(* IEC 61131-3 sources: STruCpp/tests/st-validation/function_blocks, 30 files *)

(* ---- basic_fb.st ---- *)
FUNCTION_BLOCK Counter
  VAR_INPUT increment : INT; END_VAR
  VAR_OUTPUT count : INT; END_VAR
  count := count + increment;
END_FUNCTION_BLOCK

FUNCTION_BLOCK Toggle
  VAR_OUTPUT state : BOOL; END_VAR
  state := NOT state;
END_FUNCTION_BLOCK

(* ---- fb_abstract.st ---- *)
FUNCTION_BLOCK ABSTRACT Shape
  VAR_OUTPUT area : REAL; END_VAR

  METHOD PUBLIC ABSTRACT GetArea : REAL
  END_METHOD
END_FUNCTION_BLOCK

FUNCTION_BLOCK Circle EXTENDS Shape
  VAR_INPUT radius : REAL; END_VAR

  METHOD PUBLIC GetArea : REAL
    GetArea := 3.14159 * radius * radius;
  END_METHOD

  area := THIS.GetArea();
END_FUNCTION_BLOCK

(* ---- fb_accumulator.st ---- *)
FUNCTION_BLOCK AccumulatorFB
  VAR_INPUT inc : INT; END_VAR
  VAR total : INT; END_VAR
  VAR_OUTPUT result : INT; END_VAR
  total := total + inc;
  result := total;
END_FUNCTION_BLOCK

(* ---- fb_composition.st ---- *)
FUNCTION_BLOCK Sensor
  VAR_OUTPUT value : INT; END_VAR
  value := 42;
END_FUNCTION_BLOCK

FUNCTION_BLOCK Controller
  VAR
    sensor : Sensor;
    reading : INT;
    processed : BOOL;
  END_VAR
  sensor();
  reading := sensor.value;
  processed := TRUE;
END_FUNCTION_BLOCK

(* ---- fb_constructor_defaults.st ---- *)
FUNCTION_BLOCK ConfigFB
  VAR_INPUT
    maxCount : INT;
  END_VAR
  VAR_OUTPUT
    ready : BOOL;
  END_VAR
  VAR
    counter : INT;
  END_VAR
  IF counter < maxCount THEN
    counter := counter + 1;
  END_IF;
  ready := counter >= maxCount;
END_FUNCTION_BLOCK

(* ---- fb_deep_method.st ---- *)
FUNCTION_BLOCK Inner
  VAR_INPUT seed : INT; END_VAR
  VAR_OUTPUT val : INT; END_VAR
  METHOD PUBLIC GetVal : INT
    GetVal := val + seed;
  END_METHOD
END_FUNCTION_BLOCK

FUNCTION_BLOCK Outer
  VAR
    m : Inner;
    cached : INT;
  END_VAR
  METHOD PUBLIC ReadInner : INT
    ReadInner := m.GetVal();
  END_METHOD
END_FUNCTION_BLOCK

(* ---- fb_final.st ---- *)
FUNCTION_BLOCK FINAL SealedFB
  VAR_INPUT x : INT; END_VAR
  VAR_OUTPUT y : INT; END_VAR
  y := x + 1;
END_FUNCTION_BLOCK

(* ---- fb_inheritance.st ---- *)
FUNCTION_BLOCK Base
  VAR
    _val : INT;
  END_VAR

  METHOD PUBLIC SetValue
    VAR_INPUT v : INT; END_VAR
    _val := v;
  END_METHOD

  METHOD PUBLIC GetValue : INT
    GetValue := _val;
  END_METHOD
END_FUNCTION_BLOCK

FUNCTION_BLOCK Derived EXTENDS Base
  METHOD PUBLIC DoubleIt
    _val := _val * 2;
  END_METHOD
END_FUNCTION_BLOCK

FUNCTION_BLOCK TagBase
  METHOD PUBLIC GetTag : INT
    GetTag := 1;
  END_METHOD
END_FUNCTION_BLOCK

FUNCTION_BLOCK TagDerived EXTENDS TagBase
  METHOD PUBLIC OVERRIDE GetTag : INT
    GetTag := 42;
  END_METHOD
END_FUNCTION_BLOCK

(* ---- fb_interfaces.st ---- *)
INTERFACE IMovable
  METHOD MoveTo : BOOL
    VAR_INPUT x : INT; y : INT; END_VAR
  END_METHOD
END_INTERFACE

FUNCTION_BLOCK Robot IMPLEMENTS IMovable
  VAR
    posX : INT;
    posY : INT;
  END_VAR

  METHOD MoveTo : BOOL
    VAR_INPUT x : INT; y : INT; END_VAR
    posX := x;
    posY := y;
    MoveTo := TRUE;
  END_METHOD
END_FUNCTION_BLOCK

(* ---- fb_method_collision.st ---- *)
FUNCTION_BLOCK Adder
  VAR_INPUT x : INT; END_VAR
  METHOD PUBLIC Compute : INT
    Compute := x + 100;
  END_METHOD
END_FUNCTION_BLOCK

FUNCTION_BLOCK Doubler
  VAR_INPUT x : INT; END_VAR
  METHOD PUBLIC Compute : INT
    Compute := x * 2;
  END_METHOD
END_FUNCTION_BLOCK

(* ---- fb_methods.st ---- *)
FUNCTION_BLOCK Motor
  VAR
    _speed : INT;
    _running : BOOL;
  END_VAR

  METHOD PUBLIC Start
    _running := TRUE;
  END_METHOD

  METHOD PUBLIC Stop
    _running := FALSE;
    _speed := 0;
  END_METHOD

  METHOD PUBLIC SetSpeed
    VAR_INPUT newSpeed : INT; END_VAR
    IF _running THEN
      _speed := newSpeed;
    END_IF;
  END_METHOD

  METHOD PUBLIC GetSpeed : INT
    GetSpeed := _speed;
  END_METHOD

  METHOD PUBLIC IsRunning : BOOL
    IsRunning := _running;
  END_METHOD
END_FUNCTION_BLOCK

(* ---- fb_output_capture.st ---- *)
FUNCTION_BLOCK Calculator
  VAR_INPUT a : INT; b : INT; END_VAR
  VAR_OUTPUT sum : INT; product : INT; END_VAR
  sum := a + b;
  product := a * b;
END_FUNCTION_BLOCK

(* ---- fb_properties.st ---- *)
FUNCTION_BLOCK MotorProp
  VAR _speed : INT; END_VAR

  PROPERTY Speed : INT
    GET
      Speed := _speed;
    END_GET
    SET
      IF Speed > 100 THEN
        _speed := 100;
      ELSE
        _speed := Speed;
      END_IF;
    END_SET
  END_PROPERTY
END_FUNCTION_BLOCK

FUNCTION_BLOCK ControllerProp
  VAR motor : MotorProp; END_VAR
END_FUNCTION_BLOCK

(* ---- fb_state.st ---- *)
FUNCTION_BLOCK Accumulator
  VAR_INPUT value : INT; END_VAR
  VAR_OUTPUT total : INT; END_VAR
  VAR callCount : INT; END_VAR
  total := total + value;
  callCount := callCount + 1;
END_FUNCTION_BLOCK

FUNCTION_BLOCK MaxTracker
  VAR_INPUT input : INT; END_VAR
  VAR_OUTPUT maxValue : INT; END_VAR
  IF input > maxValue THEN
    maxValue := input;
  END_IF;
END_FUNCTION_BLOCK

(* ---- fb_this_super.st ---- *)
FUNCTION_BLOCK ComputeBase
  VAR_INPUT value : INT; END_VAR
  VAR_OUTPUT result : INT; END_VAR

  METHOD PUBLIC Compute : INT
    Compute := value * 2;
  END_METHOD

  result := THIS.Compute();
END_FUNCTION_BLOCK

(* ---- test_basic_fb.st ---- *)
TEST 'Counter increments by specified amount'
  VAR c : Counter; END_VAR
  c(increment := 5);
  ASSERT_EQ(c.count, 5);
  c(increment := 3);
  ASSERT_EQ(c.count, 8);
END_TEST

TEST 'Counter starts at zero'
  VAR c : Counter; END_VAR
  ASSERT_EQ(c.count, 0);
END_TEST

TEST 'Two counters are independent'
  VAR a : Counter; b : Counter; END_VAR
  a(increment := 10);
  b(increment := 20);
  ASSERT_EQ(a.count, 10);
  ASSERT_EQ(b.count, 20);
END_TEST

TEST 'Toggle alternates state'
  VAR t : Toggle; END_VAR
  ASSERT_FALSE(t.state);
  t();
  ASSERT_TRUE(t.state);
  t();
  ASSERT_FALSE(t.state);
  t();
  ASSERT_TRUE(t.state);
END_TEST

(* ---- test_fb_abstract.st ---- *)
TEST 'Concrete class computes area'
  VAR c : Circle; END_VAR
  c(radius := 2.0);
  ASSERT_NEAR(c.area, 12.566, 0.01);
END_TEST

(* ---- test_fb_accumulator.st ---- *)
TEST 'Accumulator preserves state across calls'
  VAR acc : AccumulatorFB; END_VAR
  acc(inc := 3);
  ASSERT_EQ(acc.result, 3);
  acc(inc := 3);
  ASSERT_EQ(acc.result, 6);
  acc(inc := 3);
  ASSERT_EQ(acc.result, 9);
END_TEST

(* ---- test_fb_composition.st ---- *)
TEST 'FB composition: Controller reads Sensor'
  VAR ctrl : Controller; END_VAR
  ctrl();
  ASSERT_EQ(ctrl.reading, 42);
  ASSERT_TRUE(ctrl.processed);
END_TEST

TEST 'FB composition: nested FB invoked'
  VAR ctrl : Controller; END_VAR
  ctrl();
  ASSERT_EQ(ctrl.sensor.value, 42);
END_TEST

(* ---- test_fb_constructor_defaults.st ---- *)
TEST 'FB input not ready after single call with high limit'
  VAR cfg : ConfigFB; END_VAR
  cfg(maxCount := 100);
  ASSERT_FALSE(cfg.ready);
END_TEST

TEST 'FB input ready when limit is 1'
  VAR cfg : ConfigFB; END_VAR
  cfg(maxCount := 1);
  ASSERT_TRUE(cfg.ready);
END_TEST

(* ---- test_fb_deep_method.st ---- *)
TEST 'Method in Outer calls Inner.GetVal()'
  VAR ctrl : Outer; result : INT; END_VAR
  ctrl.m.seed := 10;
  ctrl.m.val := 5;
  result := ctrl.ReadInner();
  ASSERT_EQ(result, 15);
END_TEST

(* ---- test_fb_final.st ---- *)
TEST 'FINAL FB computes correctly'
  VAR s : SealedFB; END_VAR
  s(x := 42);
  ASSERT_EQ(s.y, 43);
END_TEST

(* ---- test_fb_inheritance.st ---- *)
TEST 'Derived inherits base methods'
  VAR d : Derived; END_VAR
  d.SetValue(v := 10);
  ASSERT_EQ(d.GetValue(), 10);
END_TEST

TEST 'Derived can add new methods'
  VAR d : Derived; END_VAR
  d.SetValue(v := 5);
  d.DoubleIt();
  ASSERT_EQ(d.GetValue(), 10);
END_TEST

TEST 'Override dispatch returns derived value'
  VAR d : TagDerived; result : INT; END_VAR
  result := d.GetTag();
  ASSERT_EQ(result, 42);
END_TEST

(* ---- test_fb_interfaces.st ---- *)
TEST 'FB implements interface method'
  VAR bot : Robot; ok : BOOL; END_VAR
  ok := bot.MoveTo(x := 10, y := 20);
  ASSERT_TRUE(ok);
  ASSERT_EQ(bot.posX, 10);
  ASSERT_EQ(bot.posY, 20);
END_TEST

(* ---- test_fb_method_collision.st ---- *)
TEST 'Two FBs with same method name dispatch correctly'
  VAR a : Adder; d : Doubler; r1, r2 : INT; END_VAR
  a.x := 5;
  d.x := 5;
  r1 := a.Compute();
  r2 := d.Compute();
  ASSERT_EQ(r1, 105);
  ASSERT_EQ(r2, 10);
END_TEST

(* ---- test_fb_methods.st ---- *)
TEST 'Motor starts and stops'
  VAR m : Motor; END_VAR
  ASSERT_FALSE(m.IsRunning());
  m.Start();
  ASSERT_TRUE(m.IsRunning());
  m.Stop();
  ASSERT_FALSE(m.IsRunning());
END_TEST

TEST 'Motor speed only changes when running'
  VAR m : Motor; END_VAR
  m.SetSpeed(newSpeed := 100);
  ASSERT_EQ(m.GetSpeed(), 0);
  m.Start();
  m.SetSpeed(newSpeed := 750);
  ASSERT_EQ(m.GetSpeed(), 750);
END_TEST

TEST 'Motor stop resets speed'
  VAR m : Motor; END_VAR
  m.Start();
  m.SetSpeed(newSpeed := 500);
  m.Stop();
  ASSERT_EQ(m.GetSpeed(), 0);
END_TEST

(* ---- test_fb_output_capture.st ---- *)
TEST 'FB output capture with => syntax'
  VAR calc : Calculator; mySum, myProduct : INT; END_VAR
  calc(a := 5, b := 3, sum => mySum, product => myProduct);
  ASSERT_EQ(mySum, 8);
  ASSERT_EQ(myProduct, 15);
END_TEST

(* ---- test_fb_properties.st ---- *)
TEST 'Property setter and getter work'
  VAR m : MotorProp; x : INT; END_VAR
  m.Speed := 75;
  x := m.Speed;
  ASSERT_EQ(x, 75);
END_TEST

TEST 'Property setter clamps above threshold'
  VAR m : MotorProp; x : INT; END_VAR
  m.Speed := 200;
  x := m.Speed;
  ASSERT_EQ(x, 100);
END_TEST

(* ---- test_fb_state.st ---- *)
TEST 'Accumulator accumulates over multiple calls'
  VAR acc : Accumulator; END_VAR
  acc(value := 10);
  acc(value := 20);
  acc(value := 30);
  ASSERT_EQ(acc.total, 60);
END_TEST

TEST 'Accumulator internal state tracks calls'
  VAR acc : Accumulator; END_VAR
  acc(value := 1);
  acc(value := 1);
  ASSERT_EQ(acc.callCount, 2);
END_TEST

TEST 'MaxTracker tracks maximum input'
  VAR mt : MaxTracker; END_VAR
  mt(input := 5);
  ASSERT_EQ(mt.maxValue, 5);
  mt(input := 3);
  ASSERT_EQ(mt.maxValue, 5);
  mt(input := 8);
  ASSERT_EQ(mt.maxValue, 8);
  mt(input := 1);
  ASSERT_EQ(mt.maxValue, 8);
END_TEST

(* ---- test_fb_this_super.st ---- *)
TEST 'Base uses THIS to call own method'
  VAR b : ComputeBase; END_VAR
  b(value := 5);
  ASSERT_EQ(b.result, 10);
END_TEST
